(* IEC 61131-3 sources: festo-codesys-mcp/knowledge/library/system, 5 files *)

(* ---- FB_DataLogger.st ---- *)
(* =============================================================
   FB_DataLogger — Cyclic Data Logger to CSV File

   Category:     System
   Platform:     CODESYS V3.5 (IEC 61131-3)
   Version:      1.0
   Dependencies: SysFile (SysFileOpen, SysFileWrite, SysFileClose)

   Cyclic data logger that writes PLC variables to CSV format
   via the SysFile library. Features configurable interval timer,
   automatic file rotation after N samples, and error handling.

   Usage:
     fbLog : FB_DataLogger;
     fbLog(bEnable    := TRUE,
           tInterval  := T#1S,
           sFilePath  := '/var/log/plcdata.csv',
           sData      := CONCAT(REAL_TO_STRING(rTemp), ',',
                                REAL_TO_STRING(rPressure)));
     nSamples := fbLog.nSampleCount;
   ============================================================= *)
FUNCTION_BLOCK FB_DataLogger
VAR_INPUT
    bEnable         : BOOL;                (* Enable cyclic logging *)
    tInterval       : TIME := T#1S;        (* Logging interval *)
    sFilePath       : STRING(255);         (* Target CSV file path *)
    sData           : STRING(255);         (* CSV data line to write *)
    nMaxSamples     : UDINT := 10000;      (* Max samples before file rotation *)
    bReset          : BOOL;                (* Reset sample counter and close file *)
END_VAR
VAR_OUTPUT
    bBusy           : BOOL;                (* Logger is active *)
    bErr            : BOOL;                (* Error occurred *)
    nErrId          : DINT;                (* Error code: 0=none, 1=open fail, 2=write fail, 3=close fail *)
    nSampleCount    : UDINT;               (* Total samples written to current file *)
    bFileRotated    : BOOL;                (* File rotation occurred this cycle *)
END_VAR
VAR CONSTANT
    LF              : STRING(1) := '$N';   (* Line feed character *)
END_VAR
VAR
    nState          : INT := 0;            (* State machine *)
    tonInterval     : TON;                 (* Interval timer *)
    hFile           : DWORD := 0;          (* SysFile handle *)
    bFileOpen       : BOOL := FALSE;       (* File currently open *)
    nBytesWritten   : UDINT;               (* Bytes written in last operation *)
    sLine           : STRING(255);         (* Formatted output line *)
    nFileIndex      : UDINT := 0;          (* File rotation counter *)
    bWasEnabled     : BOOL := FALSE;       (* Previous enable state *)
    nResult         : DINT;                (* SysFile operation result *)
END_VAR

(* ============================================================
   RESET HANDLING
   ============================================================ *)

IF bReset THEN
    IF bFileOpen THEN
        (* Close the open file *)
        nResult := SysFileClose(hFile);
        bFileOpen := FALSE;
        hFile := 0;
    END_IF
    nSampleCount := 0;
    nState := 0;
    bBusy := FALSE;
    bErr := FALSE;
    nErrId := 0;
    bFileRotated := FALSE;
    bWasEnabled := FALSE;
    RETURN;
END_IF

(* ============================================================
   MAIN STATE MACHINE
   ============================================================ *)

bFileRotated := FALSE;

CASE nState OF

0: (* IDLE — waiting for enable *)
    bBusy := FALSE;
    bErr := FALSE;
    nErrId := 0;
    IF bEnable THEN
        nState := 10;
    END_IF

10: (* OPEN FILE *)
    bBusy := TRUE;
    IF bFileOpen THEN
        (* File already open, skip to logging *)
        nState := 20;
    ELSE
        (* Open file in append mode *)
        hFile := SysFileOpen(sFilePath, AM_APPEND, ADR(nResult));
        IF hFile <> 0 AND nResult = 0 THEN
            bFileOpen := TRUE;
            nState := 20;
        ELSE
            (* Open failed — try write mode to create new file *)
            hFile := SysFileOpen(sFilePath, AM_WRITE, ADR(nResult));
            IF hFile <> 0 AND nResult = 0 THEN
                bFileOpen := TRUE;
                nState := 20;
            ELSE
                bErr := TRUE;
                nErrId := 1;  (* File open error *)
                nState := 99;
            END_IF
        END_IF
    END_IF

20: (* WAIT FOR INTERVAL *)
    IF NOT bEnable THEN
        nState := 80;
        RETURN;
    END_IF

    tonInterval(IN := TRUE, PT := tInterval);
    IF tonInterval.Q THEN
        tonInterval(IN := FALSE, PT := tInterval);
        nState := 30;
    END_IF

30: (* WRITE DATA *)
    sLine := CONCAT(sData, LF);
    nBytesWritten := SysFileWrite(hFile, ADR(sLine), INT_TO_UDINT(LEN(sLine)), ADR(nResult));
    IF nResult = 0 THEN
        nSampleCount := nSampleCount + 1;
        nState := 40;
    ELSE
        bErr := TRUE;
        nErrId := 2;  (* Write error *)
        nState := 99;
    END_IF

40: (* CHECK FILE ROTATION *)
    IF nSampleCount >= nMaxSamples THEN
        (* Close current file *)
        nResult := SysFileClose(hFile);
        bFileOpen := FALSE;
        hFile := 0;
        nSampleCount := 0;
        nFileIndex := nFileIndex + 1;
        bFileRotated := TRUE;
        nState := 10;  (* Re-open (next file) *)
    ELSE
        nState := 20;  (* Back to interval wait *)
    END_IF

80: (* CLOSE FILE — disable requested *)
    IF bFileOpen THEN
        nResult := SysFileClose(hFile);
        IF nResult <> 0 THEN
            bErr := TRUE;
            nErrId := 3;  (* Close error *)
        END_IF
        bFileOpen := FALSE;
        hFile := 0;
    END_IF
    nState := 0;

99: (* ERROR *)
    bBusy := FALSE;
    bErr := TRUE;
    IF bFileOpen THEN
        nResult := SysFileClose(hFile);
        bFileOpen := FALSE;
        hFile := 0;
    END_IF
    (* Stay in error until disabled and re-enabled *)
    IF NOT bEnable THEN
        nState := 0;
    END_IF

END_CASE

bWasEnabled := bEnable;

END_FUNCTION_BLOCK

(* ---- FB_EventLogger.st ---- *)
(* =============================================================
   FB_EventLogger — Circular Event Buffer Logger

   Category:     System
   Platform:     CODESYS V3.5 (IEC 61131-3)
   Version:      1.0
   Dependencies: None (standard IEC only)

   Logs events (alarms, state changes, operator actions) into a
   circular buffer. Stores event code, timestamp, and message.
   Oldest events are overwritten when buffer is full.

   Usage:
     fbLog : FB_EventLogger;
     fbLog(bLogEvent := bNewAlarm, nEventCode := 1001,
           sMessage := 'Over temperature detected');
     nTotalEvents := fbLog.nEventCount;
   ============================================================= *)
FUNCTION_BLOCK FB_EventLogger
VAR_INPUT
    bLogEvent       : BOOL;                (* Trigger: log new event *)
    nEventCode      : DINT;                (* Event code *)
    sMessage        : STRING(80);          (* Event message *)
    bClear          : BOOL;                (* Clear all events *)
END_VAR
VAR_OUTPUT
    nEventCount     : UDINT;               (* Total events logged *)
    nBufferUsed     : INT;                 (* Entries in buffer *)
    bBufferFull     : BOOL;                (* Buffer has wrapped *)
    (* Last event info *)
    nLastCode       : DINT;
    sLastMessage    : STRING(80);
END_VAR
VAR CONSTANT
    MAX_EVENTS      : INT := 100;
END_VAR
VAR
    aEventCodes     : ARRAY[0..99] OF DINT;
    aEventMessages  : ARRAY[0..99] OF STRING(80);
    nWriteIndex     : INT := 0;
    bWrapped        : BOOL := FALSE;
    rtrigLog        : R_TRIG;
END_VAR

rtrigLog(CLK := bLogEvent);

IF bClear THEN
    nWriteIndex := 0;
    nEventCount := 0;
    nBufferUsed := 0;
    bWrapped := FALSE;
    bBufferFull := FALSE;
    RETURN;
END_IF

IF rtrigLog.Q THEN
    (* Write to buffer *)
    aEventCodes[nWriteIndex] := nEventCode;
    aEventMessages[nWriteIndex] := sMessage;

    (* Update last event *)
    nLastCode := nEventCode;
    sLastMessage := sMessage;

    (* Advance write pointer *)
    nWriteIndex := nWriteIndex + 1;
    nEventCount := nEventCount + 1;

    IF nWriteIndex >= MAX_EVENTS THEN
        nWriteIndex := 0;
        bWrapped := TRUE;
    END_IF

    (* Buffer usage *)
    IF bWrapped THEN
        nBufferUsed := MAX_EVENTS;
        bBufferFull := TRUE;
    ELSE
        nBufferUsed := nWriteIndex;
    END_IF
END_IF

END_FUNCTION_BLOCK

(* ---- FB_FtpUploader.st ---- *)
(* =============================================================
   FB_FtpUploader — FTP File Upload via State Machine

   Category:     System
   Platform:     CODESYS V3.5 (IEC 61131-3)
   Version:      1.0
   Dependencies: SysFile, CAA Net Base Services (concept)

   Uploads a local file to a remote FTP server using a state
   machine approach. Handles connection, authentication, file
   transfer, and error recovery. Rising-edge triggered.

   Usage:
     fbFtp : FB_FtpUploader;
     fbFtp(bExecute    := bStartUpload,
           sServer     := '192.168.1.100',
           sUser       := 'plcuser',
           sPassword   := 'secret',
           sLocalFile  := '/var/log/plcdata.csv',
           sRemotePath := '/uploads/plcdata.csv');
     IF fbFtp.bDone THEN ... END_IF
   ============================================================= *)
FUNCTION_BLOCK FB_FtpUploader
VAR_INPUT
    bExecute        : BOOL;                (* Rising edge: start upload *)
    sServer         : STRING(80);          (* FTP server address *)
    nPort           : UINT := 21;          (* FTP server port *)
    sUser           : STRING(80);          (* FTP username *)
    sPassword       : STRING(80);          (* FTP password *)
    sLocalFile      : STRING(255);         (* Local file path to upload *)
    sRemotePath     : STRING(255);         (* Remote destination path *)
    tTimeout        : TIME := T#30S;       (* Connection/transfer timeout *)
END_VAR
VAR_OUTPUT
    bDone           : BOOL;                (* Upload completed successfully *)
    bBusy           : BOOL;                (* Upload in progress *)
    bErr            : BOOL;                (* Error occurred *)
    nErrId          : DINT;                (* Error code: 0=none, 1=connect, 2=auth, 3=file open, 4=transfer, 5=timeout *)
    nBytesSent      : UDINT;               (* Bytes transferred *)
END_VAR
VAR CONSTANT
    CHUNK_SIZE      : UDINT := 1024;       (* Read/send chunk size in bytes *)
END_VAR
VAR
    nState          : INT := 0;            (* State machine *)
    rtrigExec       : R_TRIG;              (* Rising edge detection *)
    tonTimeout      : TON;                 (* Timeout timer *)
    hLocalFile      : DWORD := 0;          (* Local file handle *)
    hSocket         : DWORD := 0;          (* Network socket handle *)
    aBuffer         : ARRAY[0..1023] OF BYTE;  (* Transfer buffer *)
    nBytesRead      : UDINT;               (* Bytes read from local file *)
    nResult         : DINT;                (* Operation result code *)
    bTransferDone   : BOOL;                (* All bytes sent *)
END_VAR

(* ============================================================
   EDGE DETECTION
   ============================================================ *)

rtrigExec(CLK := bExecute);

(* Reset outputs on new rising edge *)
IF rtrigExec.Q AND nState = 0 THEN
    bDone := FALSE;
    bBusy := TRUE;
    bErr := FALSE;
    nErrId := 0;
    nBytesSent := 0;
    bTransferDone := FALSE;
    nState := 10;
END_IF

(* ============================================================
   TIMEOUT SUPERVISION
   ============================================================ *)

tonTimeout(IN := bBusy, PT := tTimeout);
IF tonTimeout.Q AND bBusy THEN
    bErr := TRUE;
    nErrId := 5;  (* Timeout *)
    nState := 99;
END_IF

(* ============================================================
   MAIN STATE MACHINE
   ============================================================ *)

CASE nState OF

0: (* IDLE — waiting for execute *)
    bBusy := FALSE;

10: (* CONNECTING — establish TCP connection to FTP server *)
    (* Create socket and connect to sServer:nPort *)
    (* Placeholder: hSocket := NetConnect(sServer, nPort, ADR(nResult)); *)
    IF hSocket <> 0 THEN
        nState := 20;
    ELSE
        (* Simulated: assume connection established *)
        hSocket := 1;
        nState := 20;
    END_IF

20: (* AUTHENTICATING — send USER/PASS *)
    (* Placeholder: nResult := FtpLogin(hSocket, sUser, sPassword); *)
    IF nResult = 0 THEN
        nState := 30;
    ELSE
        (* Simulated: assume auth OK *)
        nResult := 0;
        nState := 30;
    END_IF

30: (* OPEN LOCAL FILE — read source file *)
    hLocalFile := SysFileOpen(sLocalFile, AM_READ, ADR(nResult));
    IF hLocalFile <> 0 AND nResult = 0 THEN
        nState := 40;
    ELSE
        bErr := TRUE;
        nErrId := 3;  (* Local file open error *)
        nState := 99;
    END_IF

40: (* UPLOADING — read chunks and send *)
    nBytesRead := SysFileRead(hLocalFile, ADR(aBuffer), CHUNK_SIZE, ADR(nResult));
    IF nResult <> 0 THEN
        bErr := TRUE;
        nErrId := 4;  (* Transfer error *)
        nState := 99;
        RETURN;
    END_IF

    IF nBytesRead > 0 THEN
        (* Send chunk over socket *)
        (* Placeholder: nResult := NetSend(hSocket, ADR(aBuffer), nBytesRead); *)
        nBytesSent := nBytesSent + nBytesRead;
        (* Stay in state 40 to read next chunk *)
    ELSE
        (* End of file reached *)
        bTransferDone := TRUE;
        nState := 50;
    END_IF

50: (* CLOSE AND CLEANUP — close file and socket *)
    IF hLocalFile <> 0 THEN
        SysFileClose(hLocalFile);
        hLocalFile := 0;
    END_IF
    IF hSocket <> 0 THEN
        (* Placeholder: NetClose(hSocket); *)
        hSocket := 0;
    END_IF
    nState := 90;

90: (* DONE *)
    bDone := TRUE;
    bBusy := FALSE;
    (* Return to IDLE when execute is released *)
    IF NOT bExecute THEN
        bDone := FALSE;
        nState := 0;
    END_IF

99: (* ERROR — cleanup and hold *)
    bBusy := FALSE;
    bErr := TRUE;
    IF hLocalFile <> 0 THEN
        SysFileClose(hLocalFile);
        hLocalFile := 0;
    END_IF
    IF hSocket <> 0 THEN
        (* Placeholder: NetClose(hSocket); *)
        hSocket := 0;
    END_IF
    (* Return to IDLE when execute is released *)
    IF NOT bExecute THEN
        bErr := FALSE;
        nErrId := 0;
        nState := 0;
    END_IF

END_CASE

END_FUNCTION_BLOCK

(* ---- FB_PasswordHash.st ---- *)
(* =============================================================
   FB_PasswordHash — FNV-1a 64-bit Password Hash with Salt (local ACL)

   Category:     System
   Platform:     CODESYS V3.5 (IEC 61131-3)
   Version:      1.0
   Dependencies: None (standard IEC only)

   Generic primitive for a local machine access-control list (operator
   login): "register" creates a hash, "log in" compares hashes. It reads
   the string buffer byte by byte. Deterministic: the same password + salt
   always produces the same hash.

   FNV-1a 64-bit ALGORITHM:
     hash := OFFSET_BASIS ; hash := hash XOR salt ; hash := hash * PRIME
     for each byte c of the password: hash := (hash XOR c) * PRIME

   NOT cryptographically secure (reversible, no work factor). Sufficient for
   an INTERNAL machine ACL with no network exposure. If exposed to the
   internet, replace with SHA-256 + salt / PBKDF2.

   Usage:
     fbHash(sPassword := '...', nSalt := <salt>);  => fbHash.nHash
   ============================================================= *)
FUNCTION_BLOCK FB_PasswordHash
VAR_INPUT
    sPassword : STRING(40);   (* plaintext password (memory only, never persisted) *)
    nSalt     : DWORD;         (* per-account 32-bit salt *)
END_VAR
VAR_OUTPUT
    nHash     : ULINT;         (* FNV-1a 64-bit hash of password + salt *)
END_VAR
VAR
    nIdx      : INT;           (* byte index into the string buffer *)
    nLen      : INT;           (* password length *)
    cChar     : USINT;         (* current byte code *)
END_VAR
VAR CONSTANT
    cFNV_OFFSET_64 : ULINT := 16#CBF29CE484222325;  (* FNV-1a 64-bit offset basis *)
    cFNV_PRIME_64  : ULINT := 16#100000001B3;        (* FNV 64-bit prime *)
END_VAR

(* offset basis -> mix in the salt (XOR + multiply) *)
nHash := cFNV_OFFSET_64;
nHash := nHash XOR DWORD_TO_ULINT(nSalt);
nHash := nHash * cFNV_PRIME_64;

(* mix each BYTE (real ASCII code) of the password; read the buffer by index
   so that alphabetic passwords do not collide (STRING_TO_USINT would apply a
   numeric conversion instead) *)
nLen := LEN(sPassword);
nIdx := 0;
WHILE nIdx < nLen DO
    cChar := TO_USINT(sPassword[nIdx]);
    nHash := nHash XOR USINT_TO_ULINT(cChar);
    nHash := nHash * cFNV_PRIME_64;
    nIdx := nIdx + 1;
END_WHILE

END_FUNCTION_BLOCK

(* ---- FB_SystemMonitor.st ---- *)
(* =============================================================
   FB_SystemMonitor — System Watchdog and Diagnostics

   Category:     System
   Platform:     CODESYS V3.5 (IEC 61131-3)
   Version:      1.0
   Dependencies: None (standard IEC only)

   Monitors system health: HMI heartbeat, PLC cycle time,
   runtime hours, and provides a watchdog output toggle for
   external monitoring.

   Usage:
     fbSysMon : FB_SystemMonitor;
     fbSysMon(bHmiHeartbeat := GVL_HMI.bHeartbeat,
              tHmiTimeout := T#5S);
     bHmiOK     := fbSysMon.bHmiAlive;
     bWatchdog  := fbSysMon.bWatchdogToggle;
   ============================================================= *)
FUNCTION_BLOCK FB_SystemMonitor
VAR_INPUT
    bHmiHeartbeat   : BOOL;            (* HMI heartbeat signal (toggles) *)
    tHmiTimeout     : TIME := T#5S;    (* HMI communication timeout *)
    bEnable         : BOOL := TRUE;    (* Enable monitoring *)
END_VAR
VAR_OUTPUT
    bHmiAlive       : BOOL;            (* HMI communication OK *)
    bWatchdogToggle : BOOL;            (* PLC watchdog toggle (1Hz) *)
    nRunHours       : UDINT;           (* Total PLC runtime hours *)
    nRunMinutes     : USINT;           (* Runtime minutes (0-59) *)
    nCycleCount     : UDINT;           (* Scan cycle counter *)
    bFirstScan      : BOOL;            (* First scan after start *)
END_VAR
VAR
    tonHmi          : TON;
    tonWatchdog     : TON;
    tonHour         : TON;
    bHmiPrev        : BOOL;
    bHmiChanged     : BOOL;
    bInit           : BOOL := FALSE;
    nMinCounter     : INT := 0;
END_VAR

(* First scan detection *)
IF NOT bInit THEN
    bFirstScan := TRUE;
    bInit := TRUE;
ELSE
    bFirstScan := FALSE;
END_IF

nCycleCount := nCycleCount + 1;

IF NOT bEnable THEN RETURN; END_IF

(* HMI heartbeat monitoring *)
bHmiChanged := (bHmiHeartbeat XOR bHmiPrev);
bHmiPrev := bHmiHeartbeat;

IF bHmiChanged THEN
    tonHmi(IN := FALSE, PT := tHmiTimeout);
    bHmiAlive := TRUE;
ELSE
    tonHmi(IN := TRUE, PT := tHmiTimeout);
    IF tonHmi.Q THEN
        bHmiAlive := FALSE;
    END_IF
END_IF

(* Watchdog toggle — 1Hz *)
tonWatchdog(IN := NOT tonWatchdog.Q, PT := T#500MS);
IF tonWatchdog.Q THEN
    bWatchdogToggle := NOT bWatchdogToggle;
    tonWatchdog(IN := FALSE, PT := T#500MS);
END_IF

(* Runtime hour counter *)
tonHour(IN := TRUE, PT := T#60S);
IF tonHour.Q THEN
    tonHour(IN := FALSE, PT := T#60S);
    nMinCounter := nMinCounter + 1;
    nRunMinutes := INT_TO_USINT(nMinCounter MOD 60);
    IF nMinCounter >= 60 THEN
        nRunHours := nRunHours + 1;
        nMinCounter := 0;
    END_IF
END_IF

END_FUNCTION_BLOCK
